DATA_BLOCK "Call_KeyenceCheckerIV_DB"
VAR
  InsKeyenceCheckerIV3810A1 : "FB_KeyenceCheckerIV3";
  InsKeyenceCheckerIV3811A1 : "FB_KeyenceCheckerIV3";
  nIndex : Int;
END_VAR
BEGIN
END_DATA_BLOCK
